Yaskawa INFORM job: FAT2.JBI

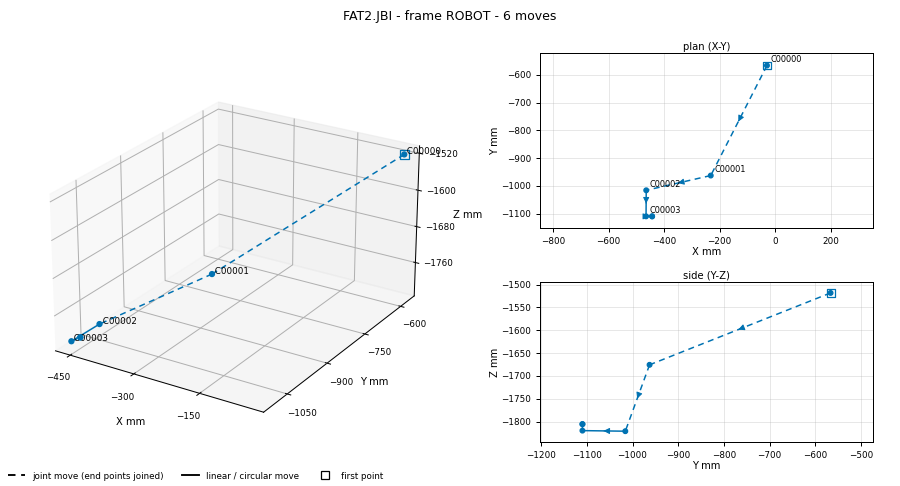
[picture p0: tool path of FAT2.JBI in frame ROBOT, 6 of 6 moves have a stored position in this frame; points joined in program order, loops and branches not executed]
/JOB
//NAME FAT2
///FOLDERNAME INNE
//POS
///NPOS 6,6,0,0,0,0
///TOOL 0
///POSTYPE ROBOT
///RECTAN
///RCONF 1,0,0,0,0,0,0,0,0,0,0,0,0,0,0,0,0,0,0,0,0,0,0,0
C00000=-29.432,-566.299,-1518.309,-40.3642,0.3679,-83.7762
C00001=-231.920,-962.701,-1675.684,-40.3495,0.3633,-83.7637
///RCONF 0,0,0,0,0,0,0,0,0,0,0,0,0,0,0,0,0,0,0,0,0,0,0,0
C00002=-464.363,-1015.789,-1821.069,-40.3545,0.3778,-83.7566
C00003=-465.038,-1109.697,-1819.785,-40.3560,0.3804,-83.7523
C00004=-443.112,-1109.674,-1805.600,-40.3554,0.3814,-83.7529
C00005=-443.112,-1109.674,-1805.600,-40.3554,0.3814,-83.7529
BC00000=2343.226,229.569,1032.161
BC00001=2339.679,24.211,1032.150
BC00002=2339.679,24.211,1032.150
BC00003=2339.679,24.211,1032.150
BC00004=2339.679,24.211,1032.150
BC00005=2339.679,24.211,1032.150
//INST
///DATE 2023/11/01 18:40
///ATTR SC,RW,RJ
////FRAME ROBOT
///GROUP1 RB1,BS1
NOP
MOVJ C00000 BC00000 VJ=15.00
MOVJ C00001 BC00001 VJ=15.00
MACRO1 MJ#(0) ARGF10
MOVJ C00002 BC00002 VJ=15.00
ARCON
MOVL C00003 BC00003 V=13.3
ARCOF
TIMER T=1.00
MOVJ C00004 BC00004 VJ=15.00
MOVJ C00005 BC00005 VJ=15.00
END
